(* IEC 61131-3 sources: Industry-PLC-LLM/data/PLCBEAD_repo/PLCBEAD_PLCEmbed-main/PLC-BEAD/Source/GEB/REVERSE, 1 file *)

(* ---- REVERSE.ST ---- *)
FUNCTION REVERSE:BYTE
VAR_INPUT
	IN :	BYTE;
END_VAR

reverse := SHL(IN,7) OR SHR(IN,7) OR (ROR(IN,3) AND BYTE#2#01000100) OR (ROL(IN,3) AND BYTE#2#00100010)
	OR (SHL(IN,1) AND BYTE#2#00010000) OR (SHR(IN,1) AND BYTE#2#00001000);

END_FUNCTION

PROGRAM program0
  VAR
    LocalVar0 : BYTE;
	LocalOUT  : BYTE;
  END_VAR
  	LocalOUT := REVERSE(LocalVar0);
END_PROGRAM
